{attribute 'qualified_only'}
{attribute 'strict'}
TYPE E_OutRobotClip :
(
	clip_A		:= 0,
	clip_B		:= 1,
);
END_TYPE

(* stored: Version 1.1.0.1, ProductVersion 3.1.4024.13
   DUT E_OutRobotClip: Id {af34574c-5768-40d9-933b-383fcc881008} *)
